Universal Robots PolyScope program: Bridge_small.urp

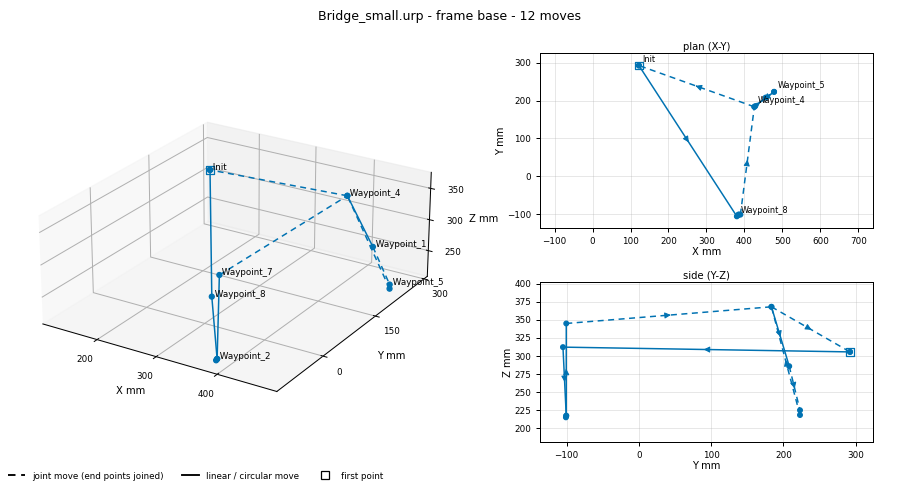
[picture p0: tool path of Bridge_small.urp in frame base, 12 of 12 moves have a stored position in this frame; points joined in program order, loops and branches not executed]
Program Bridge_small (installation=default directory=/programs/Mursal createdIn=5.11.11.1010533 lastSavedIn=5.11.11.1010533 robotSerialNumber=20205300864)
Calibrated DH parameters: a=[-0.000166, -0.243494, -0.153108, 0.000057, -0.000123, 0]; d=[0.151897, -1.34267, 53.988124, -52.514559, 0.085283, 0.092193]; alpha=[1.572472, -0.003756, 0.002824, 1.570807, -1.572621, 0]; deltaTheta=[0, 0.020704, 7.033215, -0.770746, 0.000004, 0]
Robot Program (runOnlyOnce=false)
  MoveL speed 250 mm/s, acceleration 1200 mm/s^2 (useActiveTCP=true) feature=Base
    Waypoint Init: TCP in base x=122.094 y=292.148 z=305.724 mm, rx=1.1347 ry=-2.9295 rz=0 rad; joints [91.645, -87.591, -91.764, -90.539, 90.032, 859.398] deg
    Waypoint Waypoint_8: TCP in base x=379.95 y=-105 z=312.336 mm, rx=-2.2871 ry=2.1451 rz=-0.0094 rad; joints [3.893, -107.526, -67.212, -94.674, 89.93, 720.305] deg
    Waypoint Waypoint_2: TCP in base x=385.13 y=-100.456 z=217.45 mm, rx=2.29 ry=-2.1465 rz=-0.0032 rad; joints [4.487, -111.428, -87.385, -71.283, 89.951, 720.915] deg
    Waypoint Waypoint_3: TCP in base x=383.791 y=-100.934 z=215.21 mm, rx=-2.2978 ry=2.1423 rz=0.0001 rad; joints [4.422, -111.279, -88.32, -70.297, 89.979, 720.547] deg
    URCap Gripper (Robotiq_Grippers, Robotiq Inc.) dataModel(position=100.0, force=0.7647058823529402, speed=65.0, positionInDouble=100.0, forceInDouble=0.7647058823529402, speedInDouble=65.0, slaveIds=[9], blocking=true, robotCompliant=false)
    Waypoint Waypoint_2: TCP in base x=385.13 y=-100.456 z=217.45 mm, rx=2.29 ry=-2.1465 rz=-0.0032 rad; joints [4.487, -111.428, -87.385, -71.283, 89.951, 720.915] deg
    Waypoint Waypoint_7: TCP in base x=389.341 y=-100.439 z=345.072 mm, rx=2.29 ry=-2.1465 rz=-0.0032 rad; joints [4.512, -111.773, -52.04, -106.285, 89.883, 720.869] deg
    MoveJ speed 60 deg/s, acceleration 80 deg/s^2 (useActiveTCP=true) feature=Base
      Waypoint Waypoint_4: TCP in base x=426.099 y=183.418 z=368.122 mm, rx=-2.1261 ry=2.0154 rz=-0.0437 rad; joints [39.871, -150.704, 23.3, -130.243, 89.433, 756.665] deg
    MoveL speed 250 mm/s, acceleration 1200 mm/s^2 (useActiveTCP=true) feature=Base
      Waypoint Waypoint_1: TCP in base x=456.565 y=208.029 z=285.938 mm, rx=-2.1733 ry=2.1812 rz=-0.0133 rad; joints [39.676, -142.218, -18.151, -105.918, 89.64, 759.858] deg
    MoveJ speed 60 deg/s, acceleration 80 deg/s^2 (useActiveTCP=true) feature=Base
      Waypoint Waypoint_5: TCP in base x=478.031 y=222.92 z=225.055 mm, rx=-2.226 ry=2.2168 rz=0 rad; joints [39.417, -158.302, -0.948, -110.643, 89.775, 759.115] deg
      Waypoint Waypoint_6: TCP in base x=478.034 y=222.909 z=218.422 mm, rx=2.226 ry=-2.2168 rz=0 rad; joints [39.394, -154.038, -11.761, -104.098, 89.797, 759.116] deg
      URCap Gripper (Robotiq_Grippers, Robotiq Inc.) dataModel(position=0.0, force=0.7647058823529402, speed=100.0, positionInDouble=0.0, forceInDouble=0.7647058823529402, speedInDouble=100.0, slaveIds=[9], blocking=true, robotCompliant=false)
      Waypoint Waypoint_4: TCP in base x=426.099 y=183.418 z=368.122 mm, rx=-2.1261 ry=2.0154 rz=-0.0437 rad; joints [39.871, -150.704, 23.3, -130.243, 89.433, 756.665] deg
      Waypoint Init: TCP in base x=122.094 y=292.148 z=305.724 mm, rx=1.1347 ry=-2.9295 rz=0 rad; joints [91.645, -87.591, -91.764, -90.539, 90.032, 859.398] deg
